# EPICS substitutions: gigeApp/Db/pluginTransform.substitutions
#
# pluginTransform.substitutions
#

file NDPluginBase.template
{
	{
	P=$(CAM):,
	R=Trans$(N):,
	PORT=Trans$(N),
	ADDR=0,
	TIMEOUT=1,
	NDARRAY_PORT=$(PLUGIN_PORT),
	NDARRAY_ADDR=0
	}
}

file NDTransform.template
{
	{
	P=$(CAM):,
	R=Trans$(N):,
	PORT=Trans$(N),
	ADDR=0,
	TIMEOUT=1
	}
}
